TYPE "IPC_Msg_Send_Err"
VERSION : 0.1
// Block: IPC_Msg_Send_Err
   STRUCT
      TimeOut_ACK : Bool;
      BufferShift : Struct
         Error : Bool;
         ErrCode : Int;
      END_STRUCT;
      Msg_NotAccepted : Struct
         Presence : Bool;
         Code_ACK : DInt;
         Msg : IPC_Msg_Generico;
      END_STRUCT;
   END_STRUCT;

END_TYPE
